DATA_BLOCK "DB11_INFORMES"
TITLE = DB11_INFORMES
{ S7_Optimized_Access := 'TRUE' }
AUTHOR : ABH
FAMILY : ZeusControl
VERSION : 1.0
NON_RETAIN
   VAR RETAIN
      Gestion { S7_SetPoint := 'False'} : "UDT_ZC_INF_GESTION";
      Registro { S7_SetPoint := 'False'} : "UDT_ZC_INF_DATOS";
      Buffer { S7_SetPoint := 'False'} : Array[0.."N_MAX_INF_BUFFER"] of "UDT_ZC_INF_DATOS";
   END_VAR


BEGIN
   Gestion.HabilitacionGeneral := TRUE;
   Gestion.EstadoConexion := TRUE;
   Gestion.OrdenIniciar := FALSE;
   Gestion.Etapa := 0;
   Gestion.SP_Tiempo := 10;
   Gestion.TiempoActual := 0;
   Gestion.NumeroMaxIntentos := 3;
   Gestion.Aviso.Registrar := FALSE;
   Gestion.Aviso.Estado := 0;
   Gestion.Aviso.NumeroIntentosActual := 0;
   Gestion.Datos.Registrar := 0;
   Gestion.Datos.Id := '';
   Gestion.Datos.Tipo := 0;
   Gestion.Datos.Codigo := '';
   Gestion.Datos.Fecha_1.Ano := 0;
   Gestion.Datos.Fecha_1.Mes := 0;
   Gestion.Datos.Fecha_1.Dia := 0;
   Gestion.Datos.Fecha_1.DiaSemana := 0;
   Gestion.Datos.Fecha_1.Hora := 0;
   Gestion.Datos.Fecha_1.Minuto := 0;
   Gestion.Datos.Fecha_1.Segundo := 0;
   Gestion.Datos.Fecha_1.NanoSegundo := 0;
   Gestion.Datos.Fecha_2.Ano := 0;
   Gestion.Datos.Fecha_2.Mes := 0;
   Gestion.Datos.Fecha_2.Dia := 0;
   Gestion.Datos.Fecha_2.DiaSemana := 0;
   Gestion.Datos.Fecha_2.Hora := 0;
   Gestion.Datos.Fecha_2.Minuto := 0;
   Gestion.Datos.Fecha_2.Segundo := 0;
   Gestion.Datos.Fecha_2.NanoSegundo := 0;
   Gestion.Datos.Fecha_3.Ano := 0;
   Gestion.Datos.Fecha_3.Mes := 0;
   Gestion.Datos.Fecha_3.Dia := 0;
   Gestion.Datos.Fecha_3.DiaSemana := 0;
   Gestion.Datos.Fecha_3.Hora := 0;
   Gestion.Datos.Fecha_3.Minuto := 0;
   Gestion.Datos.Fecha_3.Segundo := 0;
   Gestion.Datos.Fecha_3.NanoSegundo := 0;
   Gestion.Datos.String_1 := '';
   Gestion.Datos.String_2 := '';
   Gestion.Datos.String_3 := '';
   Gestion.Datos.String_4 := '';
   Gestion.Datos.String_5 := '';
   Gestion.Datos.String_6 := '';
   Gestion.Datos.String_7 := '';
   Gestion.Datos.String_8 := '';
   Gestion.Datos.String_9 := '';
   Gestion.Datos.String_10 := '';
   Gestion.Datos.Bool_1 := FALSE;
   Gestion.Datos.Bool_2 := FALSE;
   Gestion.Datos.Bool_3 := FALSE;
   Gestion.Datos.Bool_4 := FALSE;
   Gestion.Datos.Bool_5 := FALSE;
   Gestion.Datos.Bool_6 := FALSE;
   Gestion.Datos.Bool_7 := FALSE;
   Gestion.Datos.Bool_8 := FALSE;
   Gestion.Datos.Bool_9 := FALSE;
   Gestion.Datos.Bool_10 := FALSE;
   Gestion.Datos.Bool_11 := FALSE;
   Gestion.Datos.Bool_12 := FALSE;
   Gestion.Datos.Bool_13 := FALSE;
   Gestion.Datos.Bool_14 := FALSE;
   Gestion.Datos.Bool_15 := FALSE;
   Gestion.Datos.Bool_16 := FALSE;
   Gestion.Datos.Bool_17 := FALSE;
   Gestion.Datos.Bool_18 := FALSE;
   Gestion.Datos.Bool_19 := FALSE;
   Gestion.Datos.Bool_20 := FALSE;
   Gestion.Datos.Bool_21 := FALSE;
   Gestion.Datos.Bool_22 := FALSE;
   Gestion.Datos.Bool_23 := FALSE;
   Gestion.Datos.Bool_24 := FALSE;
   Gestion.Datos.Bool_25 := FALSE;
   Gestion.Datos.Bool_26 := FALSE;
   Gestion.Datos.Bool_27 := FALSE;
   Gestion.Datos.Bool_28 := FALSE;
   Gestion.Datos.Bool_29 := FALSE;
   Gestion.Datos.Bool_30 := FALSE;
   Gestion.Datos.Bool_31 := FALSE;
   Gestion.Datos.Bool_32 := FALSE;
   Gestion.Datos.Real_1 := 0.0;
   Gestion.Datos.Real_2 := 0.0;
   Gestion.Datos.Real_3 := 0.0;
   Gestion.Datos.Real_4 := 0.0;
   Gestion.Datos.Real_5 := 0.0;
   Gestion.Datos.Real_6 := 0.0;
   Gestion.Datos.Real_7 := 0.0;
   Gestion.Datos.Real_8 := 0.0;
   Gestion.Datos.Real_9 := 0.0;
   Gestion.Datos.Real_10 := 0.0;
   Gestion.Datos.Real_11 := 0.0;
   Gestion.Datos.Real_12 := 0.0;
   Gestion.Datos.Real_13 := 0.0;
   Gestion.Datos.Real_14 := 0.0;
   Gestion.Datos.Real_15 := 0.0;
   Gestion.Datos.Real_16 := 0.0;
   Gestion.Datos.Real_17 := 0.0;
   Gestion.Datos.Real_18 := 0.0;
   Gestion.Datos.Real_19 := 0.0;
   Gestion.Datos.Real_20 := 0.0;
   Gestion.Datos.Int_1 := 0;
   Gestion.Datos.Int_2 := 0;
   Gestion.Datos.Int_3 := 0;
   Gestion.Datos.Int_4 := 0;
   Gestion.Datos.Int_5 := 0;
   Gestion.Datos.Int_6 := 0;
   Gestion.Datos.Int_7 := 0;
   Gestion.Datos.Int_8 := 0;
   Gestion.Datos.Int_9 := 0;
   Gestion.Datos.Int_10 := 0;
   Gestion.Datos.Int_11 := 0;
   Gestion.Datos.Int_12 := 0;
   Gestion.Datos.Int_13 := 0;
   Gestion.Datos.Int_14 := 0;
   Gestion.Datos.Int_15 := 0;
   Gestion.Datos.Int_16 := 0;
   Gestion.Datos.Int_17 := 0;
   Gestion.Datos.Int_18 := 0;
   Gestion.Datos.Int_19 := 0;
   Gestion.Datos.Int_20 := 0;
   Registro.Registrar := 0;
   Registro.Id := '';
   Registro.Tipo := 0;
   Registro.Codigo := '';
   Registro.Fecha_1.Ano := 0;
   Registro.Fecha_1.Mes := 0;
   Registro.Fecha_1.Dia := 0;
   Registro.Fecha_1.DiaSemana := 0;
   Registro.Fecha_1.Hora := 0;
   Registro.Fecha_1.Minuto := 0;
   Registro.Fecha_1.Segundo := 0;
   Registro.Fecha_1.NanoSegundo := 0;
   Registro.Fecha_2.Ano := 0;
   Registro.Fecha_2.Mes := 0;
   Registro.Fecha_2.Dia := 0;
   Registro.Fecha_2.DiaSemana := 0;
   Registro.Fecha_2.Hora := 0;
   Registro.Fecha_2.Minuto := 0;
   Registro.Fecha_2.Segundo := 0;
   Registro.Fecha_2.NanoSegundo := 0;
   Registro.Fecha_3.Ano := 0;
   Registro.Fecha_3.Mes := 0;
   Registro.Fecha_3.Dia := 0;
   Registro.Fecha_3.DiaSemana := 0;
   Registro.Fecha_3.Hora := 0;
   Registro.Fecha_3.Minuto := 0;
   Registro.Fecha_3.Segundo := 0;
   Registro.Fecha_3.NanoSegundo := 0;
   Registro.String_1 := '';
   Registro.String_2 := '';
   Registro.String_3 := '';
   Registro.String_4 := '';
   Registro.String_5 := '';
   Registro.String_6 := '';
   Registro.String_7 := '';
   Registro.String_8 := '';
   Registro.String_9 := '';
   Registro.String_10 := '';
   Registro.Bool_1 := FALSE;
   Registro.Bool_2 := FALSE;
   Registro.Bool_3 := FALSE;
   Registro.Bool_4 := FALSE;
   Registro.Bool_5 := FALSE;
   Registro.Bool_6 := FALSE;
   Registro.Bool_7 := FALSE;
   Registro.Bool_8 := FALSE;
   Registro.Bool_9 := FALSE;
   Registro.Bool_10 := FALSE;
   Registro.Bool_11 := FALSE;
   Registro.Bool_12 := FALSE;
   Registro.Bool_13 := FALSE;
   Registro.Bool_14 := FALSE;
   Registro.Bool_15 := FALSE;
   Registro.Bool_16 := FALSE;
   Registro.Bool_17 := FALSE;
   Registro.Bool_18 := FALSE;
   Registro.Bool_19 := FALSE;
   Registro.Bool_20 := FALSE;
   Registro.Bool_21 := FALSE;
   Registro.Bool_22 := FALSE;
   Registro.Bool_23 := FALSE;
   Registro.Bool_24 := FALSE;
   Registro.Bool_25 := FALSE;
   Registro.Bool_26 := FALSE;
   Registro.Bool_27 := FALSE;
   Registro.Bool_28 := FALSE;
   Registro.Bool_29 := FALSE;
   Registro.Bool_30 := FALSE;
   Registro.Bool_31 := FALSE;
   Registro.Bool_32 := FALSE;
   Registro.Real_1 := 0.0;
   Registro.Real_2 := 0.0;
   Registro.Real_3 := 0.0;
   Registro.Real_4 := 0.0;
   Registro.Real_5 := 0.0;
   Registro.Real_6 := 0.0;
   Registro.Real_7 := 0.0;
   Registro.Real_8 := 0.0;
   Registro.Real_9 := 0.0;
   Registro.Real_10 := 0.0;
   Registro.Real_11 := 0.0;
   Registro.Real_12 := 0.0;
   Registro.Real_13 := 0.0;
   Registro.Real_14 := 0.0;
   Registro.Real_15 := 0.0;
   Registro.Real_16 := 0.0;
   Registro.Real_17 := 0.0;
   Registro.Real_18 := 0.0;
   Registro.Real_19 := 0.0;
   Registro.Real_20 := 0.0;
   Registro.Int_1 := 0;
   Registro.Int_2 := 0;
   Registro.Int_3 := 0;
   Registro.Int_4 := 0;
   Registro.Int_5 := 0;
   Registro.Int_6 := 0;
   Registro.Int_7 := 0;
   Registro.Int_8 := 0;
   Registro.Int_9 := 0;
   Registro.Int_10 := 0;
   Registro.Int_11 := 0;
   Registro.Int_12 := 0;
   Registro.Int_13 := 0;
   Registro.Int_14 := 0;
   Registro.Int_15 := 0;
   Registro.Int_16 := 0;
   Registro.Int_17 := 0;
   Registro.Int_18 := 0;
   Registro.Int_19 := 0;
   Registro.Int_20 := 0;
   Buffer[0].Registrar := 0;
   Buffer[0].Id := '';
   Buffer[0].Tipo := 0;
   Buffer[0].Codigo := '';
   Buffer[0].Fecha_1.Ano := 0;
   Buffer[0].Fecha_1.Mes := 0;
   Buffer[0].Fecha_1.Dia := 0;
   Buffer[0].Fecha_1.DiaSemana := 0;
   Buffer[0].Fecha_1.Hora := 0;
   Buffer[0].Fecha_1.Minuto := 0;
   Buffer[0].Fecha_1.Segundo := 0;
   Buffer[0].Fecha_1.NanoSegundo := 0;
   Buffer[0].Fecha_2.Ano := 0;
   Buffer[0].Fecha_2.Mes := 0;
   Buffer[0].Fecha_2.Dia := 0;
   Buffer[0].Fecha_2.DiaSemana := 0;
   Buffer[0].Fecha_2.Hora := 0;
   Buffer[0].Fecha_2.Minuto := 0;
   Buffer[0].Fecha_2.Segundo := 0;
   Buffer[0].Fecha_2.NanoSegundo := 0;
   Buffer[0].Fecha_3.Ano := 0;
   Buffer[0].Fecha_3.Mes := 0;
   Buffer[0].Fecha_3.Dia := 0;
   Buffer[0].Fecha_3.DiaSemana := 0;
   Buffer[0].Fecha_3.Hora := 0;
   Buffer[0].Fecha_3.Minuto := 0;
   Buffer[0].Fecha_3.Segundo := 0;
   Buffer[0].Fecha_3.NanoSegundo := 0;
   Buffer[0].String_1 := '';
   Buffer[0].String_2 := '';
   Buffer[0].String_3 := '';
   Buffer[0].String_4 := '';
   Buffer[0].String_5 := '';
   Buffer[0].String_6 := '';
   Buffer[0].String_7 := '';
   Buffer[0].String_8 := '';
   Buffer[0].String_9 := '';
   Buffer[0].String_10 := '';
   Buffer[0].Bool_1 := FALSE;
   Buffer[0].Bool_2 := FALSE;
   Buffer[0].Bool_3 := FALSE;
   Buffer[0].Bool_4 := FALSE;
   Buffer[0].Bool_5 := FALSE;
   Buffer[0].Bool_6 := FALSE;
   Buffer[0].Bool_7 := FALSE;
   Buffer[0].Bool_8 := FALSE;
   Buffer[0].Bool_9 := FALSE;
   Buffer[0].Bool_10 := FALSE;
   Buffer[0].Bool_11 := FALSE;
   Buffer[0].Bool_12 := FALSE;
   Buffer[0].Bool_13 := FALSE;
   Buffer[0].Bool_14 := FALSE;
   Buffer[0].Bool_15 := FALSE;
   Buffer[0].Bool_16 := FALSE;
   Buffer[0].Bool_17 := FALSE;
   Buffer[0].Bool_18 := FALSE;
   Buffer[0].Bool_19 := FALSE;
   Buffer[0].Bool_20 := FALSE;
   Buffer[0].Bool_21 := FALSE;
   Buffer[0].Bool_22 := FALSE;
   Buffer[0].Bool_23 := FALSE;
   Buffer[0].Bool_24 := FALSE;
   Buffer[0].Bool_25 := FALSE;
   Buffer[0].Bool_26 := FALSE;
   Buffer[0].Bool_27 := FALSE;
   Buffer[0].Bool_28 := FALSE;
   Buffer[0].Bool_29 := FALSE;
   Buffer[0].Bool_30 := FALSE;
   Buffer[0].Bool_31 := FALSE;
   Buffer[0].Bool_32 := FALSE;
   Buffer[0].Real_1 := 0.0;
   Buffer[0].Real_2 := 0.0;
   Buffer[0].Real_3 := 0.0;
   Buffer[0].Real_4 := 0.0;
   Buffer[0].Real_5 := 0.0;
   Buffer[0].Real_6 := 0.0;
   Buffer[0].Real_7 := 0.0;
   Buffer[0].Real_8 := 0.0;
   Buffer[0].Real_9 := 0.0;
   Buffer[0].Real_10 := 0.0;
   Buffer[0].Real_11 := 0.0;
   Buffer[0].Real_12 := 0.0;
   Buffer[0].Real_13 := 0.0;
   Buffer[0].Real_14 := 0.0;
   Buffer[0].Real_15 := 0.0;
   Buffer[0].Real_16 := 0.0;
   Buffer[0].Real_17 := 0.0;
   Buffer[0].Real_18 := 0.0;
   Buffer[0].Real_19 := 0.0;
   Buffer[0].Real_20 := 0.0;
   Buffer[0].Int_1 := 0;
   Buffer[0].Int_2 := 0;
   Buffer[0].Int_3 := 0;
   Buffer[0].Int_4 := 0;
   Buffer[0].Int_5 := 0;
   Buffer[0].Int_6 := 0;
   Buffer[0].Int_7 := 0;
   Buffer[0].Int_8 := 0;
   Buffer[0].Int_9 := 0;
   Buffer[0].Int_10 := 0;
   Buffer[0].Int_11 := 0;
   Buffer[0].Int_12 := 0;
   Buffer[0].Int_13 := 0;
   Buffer[0].Int_14 := 0;
   Buffer[0].Int_15 := 0;
   Buffer[0].Int_16 := 0;
   Buffer[0].Int_17 := 0;
   Buffer[0].Int_18 := 0;
   Buffer[0].Int_19 := 0;
   Buffer[0].Int_20 := 0;
   Buffer[1].Registrar := 0;
   Buffer[1].Id := '';
   Buffer[1].Tipo := 0;
   Buffer[1].Codigo := '';
   Buffer[1].Fecha_1.Ano := 0;
   Buffer[1].Fecha_1.Mes := 0;
   Buffer[1].Fecha_1.Dia := 0;
   Buffer[1].Fecha_1.DiaSemana := 0;
   Buffer[1].Fecha_1.Hora := 0;
   Buffer[1].Fecha_1.Minuto := 0;
   Buffer[1].Fecha_1.Segundo := 0;
   Buffer[1].Fecha_1.NanoSegundo := 0;
   Buffer[1].Fecha_2.Ano := 0;
   Buffer[1].Fecha_2.Mes := 0;
   Buffer[1].Fecha_2.Dia := 0;
   Buffer[1].Fecha_2.DiaSemana := 0;
   Buffer[1].Fecha_2.Hora := 0;
   Buffer[1].Fecha_2.Minuto := 0;
   Buffer[1].Fecha_2.Segundo := 0;
   Buffer[1].Fecha_2.NanoSegundo := 0;
   Buffer[1].Fecha_3.Ano := 0;
   Buffer[1].Fecha_3.Mes := 0;
   Buffer[1].Fecha_3.Dia := 0;
   Buffer[1].Fecha_3.DiaSemana := 0;
   Buffer[1].Fecha_3.Hora := 0;
   Buffer[1].Fecha_3.Minuto := 0;
   Buffer[1].Fecha_3.Segundo := 0;
   Buffer[1].Fecha_3.NanoSegundo := 0;
   Buffer[1].String_1 := '';
   Buffer[1].String_2 := '';
   Buffer[1].String_3 := '';
   Buffer[1].String_4 := '';
   Buffer[1].String_5 := '';
   Buffer[1].String_6 := '';
   Buffer[1].String_7 := '';
   Buffer[1].String_8 := '';
   Buffer[1].String_9 := '';
   Buffer[1].String_10 := '';
   Buffer[1].Bool_1 := FALSE;
   Buffer[1].Bool_2 := FALSE;
   Buffer[1].Bool_3 := FALSE;
   Buffer[1].Bool_4 := FALSE;
   Buffer[1].Bool_5 := FALSE;
   Buffer[1].Bool_6 := FALSE;
   Buffer[1].Bool_7 := FALSE;
   Buffer[1].Bool_8 := FALSE;
   Buffer[1].Bool_9 := FALSE;
   Buffer[1].Bool_10 := FALSE;
   Buffer[1].Bool_11 := FALSE;
   Buffer[1].Bool_12 := FALSE;
   Buffer[1].Bool_13 := FALSE;
   Buffer[1].Bool_14 := FALSE;
   Buffer[1].Bool_15 := FALSE;
   Buffer[1].Bool_16 := FALSE;
   Buffer[1].Bool_17 := FALSE;
   Buffer[1].Bool_18 := FALSE;
   Buffer[1].Bool_19 := FALSE;
   Buffer[1].Bool_20 := FALSE;
   Buffer[1].Bool_21 := FALSE;
   Buffer[1].Bool_22 := FALSE;
   Buffer[1].Bool_23 := FALSE;
   Buffer[1].Bool_24 := FALSE;
   Buffer[1].Bool_25 := FALSE;
   Buffer[1].Bool_26 := FALSE;
   Buffer[1].Bool_27 := FALSE;
   Buffer[1].Bool_28 := FALSE;
   Buffer[1].Bool_29 := FALSE;
   Buffer[1].Bool_30 := FALSE;
   Buffer[1].Bool_31 := FALSE;
   Buffer[1].Bool_32 := FALSE;
   Buffer[1].Real_1 := 0.0;
   Buffer[1].Real_2 := 0.0;
   Buffer[1].Real_3 := 0.0;
   Buffer[1].Real_4 := 0.0;
   Buffer[1].Real_5 := 0.0;
   Buffer[1].Real_6 := 0.0;
   Buffer[1].Real_7 := 0.0;
   Buffer[1].Real_8 := 0.0;
   Buffer[1].Real_9 := 0.0;
   Buffer[1].Real_10 := 0.0;
   Buffer[1].Real_11 := 0.0;
   Buffer[1].Real_12 := 0.0;
   Buffer[1].Real_13 := 0.0;
   Buffer[1].Real_14 := 0.0;
   Buffer[1].Real_15 := 0.0;
   Buffer[1].Real_16 := 0.0;
   Buffer[1].Real_17 := 0.0;
   Buffer[1].Real_18 := 0.0;
   Buffer[1].Real_19 := 0.0;
   Buffer[1].Real_20 := 0.0;
   Buffer[1].Int_1 := 0;
   Buffer[1].Int_2 := 0;
   Buffer[1].Int_3 := 0;
   Buffer[1].Int_4 := 0;
   Buffer[1].Int_5 := 0;
   Buffer[1].Int_6 := 0;
   Buffer[1].Int_7 := 0;
   Buffer[1].Int_8 := 0;
   Buffer[1].Int_9 := 0;
   Buffer[1].Int_10 := 0;
   Buffer[1].Int_11 := 0;
   Buffer[1].Int_12 := 0;
   Buffer[1].Int_13 := 0;
   Buffer[1].Int_14 := 0;
   Buffer[1].Int_15 := 0;
   Buffer[1].Int_16 := 0;
   Buffer[1].Int_17 := 0;
   Buffer[1].Int_18 := 0;
   Buffer[1].Int_19 := 0;
   Buffer[1].Int_20 := 0;
   Buffer[2].Registrar := 0;
   Buffer[2].Id := '';
   Buffer[2].Tipo := 0;
   Buffer[2].Codigo := '';
   Buffer[2].Fecha_1.Ano := 0;
   Buffer[2].Fecha_1.Mes := 0;
   Buffer[2].Fecha_1.Dia := 0;
   Buffer[2].Fecha_1.DiaSemana := 0;
   Buffer[2].Fecha_1.Hora := 0;
   Buffer[2].Fecha_1.Minuto := 0;
   Buffer[2].Fecha_1.Segundo := 0;
   Buffer[2].Fecha_1.NanoSegundo := 0;
   Buffer[2].Fecha_2.Ano := 0;
   Buffer[2].Fecha_2.Mes := 0;
   Buffer[2].Fecha_2.Dia := 0;
   Buffer[2].Fecha_2.DiaSemana := 0;
   Buffer[2].Fecha_2.Hora := 0;
   Buffer[2].Fecha_2.Minuto := 0;
   Buffer[2].Fecha_2.Segundo := 0;
   Buffer[2].Fecha_2.NanoSegundo := 0;
   Buffer[2].Fecha_3.Ano := 0;
   Buffer[2].Fecha_3.Mes := 0;
   Buffer[2].Fecha_3.Dia := 0;
   Buffer[2].Fecha_3.DiaSemana := 0;
   Buffer[2].Fecha_3.Hora := 0;
   Buffer[2].Fecha_3.Minuto := 0;
   Buffer[2].Fecha_3.Segundo := 0;
   Buffer[2].Fecha_3.NanoSegundo := 0;
   Buffer[2].String_1 := '';
   Buffer[2].String_2 := '';
   Buffer[2].String_3 := '';
   Buffer[2].String_4 := '';
   Buffer[2].String_5 := '';
   Buffer[2].String_6 := '';
   Buffer[2].String_7 := '';
   Buffer[2].String_8 := '';
   Buffer[2].String_9 := '';
   Buffer[2].String_10 := '';
   Buffer[2].Bool_1 := FALSE;
   Buffer[2].Bool_2 := FALSE;
   Buffer[2].Bool_3 := FALSE;
   Buffer[2].Bool_4 := FALSE;
   Buffer[2].Bool_5 := FALSE;
   Buffer[2].Bool_6 := FALSE;
   Buffer[2].Bool_7 := FALSE;
   Buffer[2].Bool_8 := FALSE;
   Buffer[2].Bool_9 := FALSE;
   Buffer[2].Bool_10 := FALSE;
   Buffer[2].Bool_11 := FALSE;
   Buffer[2].Bool_12 := FALSE;
   Buffer[2].Bool_13 := FALSE;
   Buffer[2].Bool_14 := FALSE;
   Buffer[2].Bool_15 := FALSE;
   Buffer[2].Bool_16 := FALSE;
   Buffer[2].Bool_17 := FALSE;
   Buffer[2].Bool_18 := FALSE;
   Buffer[2].Bool_19 := FALSE;
   Buffer[2].Bool_20 := FALSE;
   Buffer[2].Bool_21 := FALSE;
   Buffer[2].Bool_22 := FALSE;
   Buffer[2].Bool_23 := FALSE;
   Buffer[2].Bool_24 := FALSE;
   Buffer[2].Bool_25 := FALSE;
   Buffer[2].Bool_26 := FALSE;
   Buffer[2].Bool_27 := FALSE;
   Buffer[2].Bool_28 := FALSE;
   Buffer[2].Bool_29 := FALSE;
   Buffer[2].Bool_30 := FALSE;
   Buffer[2].Bool_31 := FALSE;
   Buffer[2].Bool_32 := FALSE;
   Buffer[2].Real_1 := 0.0;
   Buffer[2].Real_2 := 0.0;
   Buffer[2].Real_3 := 0.0;
   Buffer[2].Real_4 := 0.0;
   Buffer[2].Real_5 := 0.0;
   Buffer[2].Real_6 := 0.0;
   Buffer[2].Real_7 := 0.0;
   Buffer[2].Real_8 := 0.0;
   Buffer[2].Real_9 := 0.0;
   Buffer[2].Real_10 := 0.0;
   Buffer[2].Real_11 := 0.0;
   Buffer[2].Real_12 := 0.0;
   Buffer[2].Real_13 := 0.0;
   Buffer[2].Real_14 := 0.0;
   Buffer[2].Real_15 := 0.0;
   Buffer[2].Real_16 := 0.0;
   Buffer[2].Real_17 := 0.0;
   Buffer[2].Real_18 := 0.0;
   Buffer[2].Real_19 := 0.0;
   Buffer[2].Real_20 := 0.0;
   Buffer[2].Int_1 := 0;
   Buffer[2].Int_2 := 0;
   Buffer[2].Int_3 := 0;
   Buffer[2].Int_4 := 0;
   Buffer[2].Int_5 := 0;
   Buffer[2].Int_6 := 0;
   Buffer[2].Int_7 := 0;
   Buffer[2].Int_8 := 0;
   Buffer[2].Int_9 := 0;
   Buffer[2].Int_10 := 0;
   Buffer[2].Int_11 := 0;
   Buffer[2].Int_12 := 0;
   Buffer[2].Int_13 := 0;
   Buffer[2].Int_14 := 0;
   Buffer[2].Int_15 := 0;
   Buffer[2].Int_16 := 0;
   Buffer[2].Int_17 := 0;
   Buffer[2].Int_18 := 0;
   Buffer[2].Int_19 := 0;
   Buffer[2].Int_20 := 0;
   Buffer[3].Registrar := 0;
   Buffer[3].Id := '';
   Buffer[3].Tipo := 0;
   Buffer[3].Codigo := '';
   Buffer[3].Fecha_1.Ano := 0;
   Buffer[3].Fecha_1.Mes := 0;
   Buffer[3].Fecha_1.Dia := 0;
   Buffer[3].Fecha_1.DiaSemana := 0;
   Buffer[3].Fecha_1.Hora := 0;
   Buffer[3].Fecha_1.Minuto := 0;
   Buffer[3].Fecha_1.Segundo := 0;
   Buffer[3].Fecha_1.NanoSegundo := 0;
   Buffer[3].Fecha_2.Ano := 0;
   Buffer[3].Fecha_2.Mes := 0;
   Buffer[3].Fecha_2.Dia := 0;
   Buffer[3].Fecha_2.DiaSemana := 0;
   Buffer[3].Fecha_2.Hora := 0;
   Buffer[3].Fecha_2.Minuto := 0;
   Buffer[3].Fecha_2.Segundo := 0;
   Buffer[3].Fecha_2.NanoSegundo := 0;
   Buffer[3].Fecha_3.Ano := 0;
   Buffer[3].Fecha_3.Mes := 0;
   Buffer[3].Fecha_3.Dia := 0;
   Buffer[3].Fecha_3.DiaSemana := 0;
   Buffer[3].Fecha_3.Hora := 0;
   Buffer[3].Fecha_3.Minuto := 0;
   Buffer[3].Fecha_3.Segundo := 0;
   Buffer[3].Fecha_3.NanoSegundo := 0;
   Buffer[3].String_1 := '';
   Buffer[3].String_2 := '';
   Buffer[3].String_3 := '';
   Buffer[3].String_4 := '';
   Buffer[3].String_5 := '';
   Buffer[3].String_6 := '';
   Buffer[3].String_7 := '';
   Buffer[3].String_8 := '';
   Buffer[3].String_9 := '';
   Buffer[3].String_10 := '';
   Buffer[3].Bool_1 := FALSE;
   Buffer[3].Bool_2 := FALSE;
   Buffer[3].Bool_3 := FALSE;
   Buffer[3].Bool_4 := FALSE;
   Buffer[3].Bool_5 := FALSE;
   Buffer[3].Bool_6 := FALSE;
   Buffer[3].Bool_7 := FALSE;
   Buffer[3].Bool_8 := FALSE;
   Buffer[3].Bool_9 := FALSE;
   Buffer[3].Bool_10 := FALSE;
   Buffer[3].Bool_11 := FALSE;
   Buffer[3].Bool_12 := FALSE;
   Buffer[3].Bool_13 := FALSE;
   Buffer[3].Bool_14 := FALSE;
   Buffer[3].Bool_15 := FALSE;
   Buffer[3].Bool_16 := FALSE;
   Buffer[3].Bool_17 := FALSE;
   Buffer[3].Bool_18 := FALSE;
   Buffer[3].Bool_19 := FALSE;
   Buffer[3].Bool_20 := FALSE;
   Buffer[3].Bool_21 := FALSE;
   Buffer[3].Bool_22 := FALSE;
   Buffer[3].Bool_23 := FALSE;
   Buffer[3].Bool_24 := FALSE;
   Buffer[3].Bool_25 := FALSE;
   Buffer[3].Bool_26 := FALSE;
   Buffer[3].Bool_27 := FALSE;
   Buffer[3].Bool_28 := FALSE;
   Buffer[3].Bool_29 := FALSE;
   Buffer[3].Bool_30 := FALSE;
   Buffer[3].Bool_31 := FALSE;
   Buffer[3].Bool_32 := FALSE;
   Buffer[3].Real_1 := 0.0;
   Buffer[3].Real_2 := 0.0;
   Buffer[3].Real_3 := 0.0;
   Buffer[3].Real_4 := 0.0;
   Buffer[3].Real_5 := 0.0;
   Buffer[3].Real_6 := 0.0;
   Buffer[3].Real_7 := 0.0;
   Buffer[3].Real_8 := 0.0;
   Buffer[3].Real_9 := 0.0;
   Buffer[3].Real_10 := 0.0;
   Buffer[3].Real_11 := 0.0;
   Buffer[3].Real_12 := 0.0;
   Buffer[3].Real_13 := 0.0;
   Buffer[3].Real_14 := 0.0;
   Buffer[3].Real_15 := 0.0;
   Buffer[3].Real_16 := 0.0;
   Buffer[3].Real_17 := 0.0;
   Buffer[3].Real_18 := 0.0;
   Buffer[3].Real_19 := 0.0;
   Buffer[3].Real_20 := 0.0;
   Buffer[3].Int_1 := 0;
   Buffer[3].Int_2 := 0;
   Buffer[3].Int_3 := 0;
   Buffer[3].Int_4 := 0;
   Buffer[3].Int_5 := 0;
   Buffer[3].Int_6 := 0;
   Buffer[3].Int_7 := 0;
   Buffer[3].Int_8 := 0;
   Buffer[3].Int_9 := 0;
   Buffer[3].Int_10 := 0;
   Buffer[3].Int_11 := 0;
   Buffer[3].Int_12 := 0;
   Buffer[3].Int_13 := 0;
   Buffer[3].Int_14 := 0;
   Buffer[3].Int_15 := 0;
   Buffer[3].Int_16 := 0;
   Buffer[3].Int_17 := 0;
   Buffer[3].Int_18 := 0;
   Buffer[3].Int_19 := 0;
   Buffer[3].Int_20 := 0;
   Buffer[4].Registrar := 0;
   Buffer[4].Id := '';
   Buffer[4].Tipo := 0;
   Buffer[4].Codigo := '';
   Buffer[4].Fecha_1.Ano := 0;
   Buffer[4].Fecha_1.Mes := 0;
   Buffer[4].Fecha_1.Dia := 0;
   Buffer[4].Fecha_1.DiaSemana := 0;
   Buffer[4].Fecha_1.Hora := 0;
   Buffer[4].Fecha_1.Minuto := 0;
   Buffer[4].Fecha_1.Segundo := 0;
   Buffer[4].Fecha_1.NanoSegundo := 0;
   Buffer[4].Fecha_2.Ano := 0;
   Buffer[4].Fecha_2.Mes := 0;
   Buffer[4].Fecha_2.Dia := 0;
   Buffer[4].Fecha_2.DiaSemana := 0;
   Buffer[4].Fecha_2.Hora := 0;
   Buffer[4].Fecha_2.Minuto := 0;
   Buffer[4].Fecha_2.Segundo := 0;
   Buffer[4].Fecha_2.NanoSegundo := 0;
   Buffer[4].Fecha_3.Ano := 0;
   Buffer[4].Fecha_3.Mes := 0;
   Buffer[4].Fecha_3.Dia := 0;
   Buffer[4].Fecha_3.DiaSemana := 0;
   Buffer[4].Fecha_3.Hora := 0;
   Buffer[4].Fecha_3.Minuto := 0;
   Buffer[4].Fecha_3.Segundo := 0;
   Buffer[4].Fecha_3.NanoSegundo := 0;
   Buffer[4].String_1 := '';
   Buffer[4].String_2 := '';
   Buffer[4].String_3 := '';
   Buffer[4].String_4 := '';
   Buffer[4].String_5 := '';
   Buffer[4].String_6 := '';
   Buffer[4].String_7 := '';
   Buffer[4].String_8 := '';
   Buffer[4].String_9 := '';
   Buffer[4].String_10 := '';
   Buffer[4].Bool_1 := FALSE;
   Buffer[4].Bool_2 := FALSE;
   Buffer[4].Bool_3 := FALSE;
   Buffer[4].Bool_4 := FALSE;
   Buffer[4].Bool_5 := FALSE;
   Buffer[4].Bool_6 := FALSE;
   Buffer[4].Bool_7 := FALSE;
   Buffer[4].Bool_8 := FALSE;
   Buffer[4].Bool_9 := FALSE;
   Buffer[4].Bool_10 := FALSE;
   Buffer[4].Bool_11 := FALSE;
   Buffer[4].Bool_12 := FALSE;
   Buffer[4].Bool_13 := FALSE;
   Buffer[4].Bool_14 := FALSE;
   Buffer[4].Bool_15 := FALSE;
   Buffer[4].Bool_16 := FALSE;
   Buffer[4].Bool_17 := FALSE;
   Buffer[4].Bool_18 := FALSE;
   Buffer[4].Bool_19 := FALSE;
   Buffer[4].Bool_20 := FALSE;
   Buffer[4].Bool_21 := FALSE;
   Buffer[4].Bool_22 := FALSE;
   Buffer[4].Bool_23 := FALSE;
   Buffer[4].Bool_24 := FALSE;
   Buffer[4].Bool_25 := FALSE;
   Buffer[4].Bool_26 := FALSE;
   Buffer[4].Bool_27 := FALSE;
   Buffer[4].Bool_28 := FALSE;
   Buffer[4].Bool_29 := FALSE;
   Buffer[4].Bool_30 := FALSE;
   Buffer[4].Bool_31 := FALSE;
   Buffer[4].Bool_32 := FALSE;
   Buffer[4].Real_1 := 0.0;
   Buffer[4].Real_2 := 0.0;
   Buffer[4].Real_3 := 0.0;
   Buffer[4].Real_4 := 0.0;
   Buffer[4].Real_5 := 0.0;
   Buffer[4].Real_6 := 0.0;
   Buffer[4].Real_7 := 0.0;
   Buffer[4].Real_8 := 0.0;
   Buffer[4].Real_9 := 0.0;
   Buffer[4].Real_10 := 0.0;
   Buffer[4].Real_11 := 0.0;
   Buffer[4].Real_12 := 0.0;
   Buffer[4].Real_13 := 0.0;
   Buffer[4].Real_14 := 0.0;
   Buffer[4].Real_15 := 0.0;
   Buffer[4].Real_16 := 0.0;
   Buffer[4].Real_17 := 0.0;
   Buffer[4].Real_18 := 0.0;
   Buffer[4].Real_19 := 0.0;
   Buffer[4].Real_20 := 0.0;
   Buffer[4].Int_1 := 0;
   Buffer[4].Int_2 := 0;
   Buffer[4].Int_3 := 0;
   Buffer[4].Int_4 := 0;
   Buffer[4].Int_5 := 0;
   Buffer[4].Int_6 := 0;
   Buffer[4].Int_7 := 0;
   Buffer[4].Int_8 := 0;
   Buffer[4].Int_9 := 0;
   Buffer[4].Int_10 := 0;
   Buffer[4].Int_11 := 0;
   Buffer[4].Int_12 := 0;
   Buffer[4].Int_13 := 0;
   Buffer[4].Int_14 := 0;
   Buffer[4].Int_15 := 0;
   Buffer[4].Int_16 := 0;
   Buffer[4].Int_17 := 0;
   Buffer[4].Int_18 := 0;
   Buffer[4].Int_19 := 0;
   Buffer[4].Int_20 := 0;
   Buffer[5].Registrar := 0;
   Buffer[5].Id := '';
   Buffer[5].Tipo := 0;
   Buffer[5].Codigo := '';
   Buffer[5].Fecha_1.Ano := 0;
   Buffer[5].Fecha_1.Mes := 0;
   Buffer[5].Fecha_1.Dia := 0;
   Buffer[5].Fecha_1.DiaSemana := 0;
   Buffer[5].Fecha_1.Hora := 0;
   Buffer[5].Fecha_1.Minuto := 0;
   Buffer[5].Fecha_1.Segundo := 0;
   Buffer[5].Fecha_1.NanoSegundo := 0;
   Buffer[5].Fecha_2.Ano := 0;
   Buffer[5].Fecha_2.Mes := 0;
   Buffer[5].Fecha_2.Dia := 0;
   Buffer[5].Fecha_2.DiaSemana := 0;
   Buffer[5].Fecha_2.Hora := 0;
   Buffer[5].Fecha_2.Minuto := 0;
   Buffer[5].Fecha_2.Segundo := 0;
   Buffer[5].Fecha_2.NanoSegundo := 0;
   Buffer[5].Fecha_3.Ano := 0;
   Buffer[5].Fecha_3.Mes := 0;
   Buffer[5].Fecha_3.Dia := 0;
   Buffer[5].Fecha_3.DiaSemana := 0;
   Buffer[5].Fecha_3.Hora := 0;
   Buffer[5].Fecha_3.Minuto := 0;
   Buffer[5].Fecha_3.Segundo := 0;
   Buffer[5].Fecha_3.NanoSegundo := 0;
   Buffer[5].String_1 := '';
   Buffer[5].String_2 := '';
   Buffer[5].String_3 := '';
   Buffer[5].String_4 := '';
   Buffer[5].String_5 := '';
   Buffer[5].String_6 := '';
   Buffer[5].String_7 := '';
   Buffer[5].String_8 := '';
   Buffer[5].String_9 := '';
   Buffer[5].String_10 := '';
   Buffer[5].Bool_1 := FALSE;
   Buffer[5].Bool_2 := FALSE;
   Buffer[5].Bool_3 := FALSE;
   Buffer[5].Bool_4 := FALSE;
   Buffer[5].Bool_5 := FALSE;
   Buffer[5].Bool_6 := FALSE;
   Buffer[5].Bool_7 := FALSE;
   Buffer[5].Bool_8 := FALSE;
   Buffer[5].Bool_9 := FALSE;
   Buffer[5].Bool_10 := FALSE;
   Buffer[5].Bool_11 := FALSE;
   Buffer[5].Bool_12 := FALSE;
   Buffer[5].Bool_13 := FALSE;
   Buffer[5].Bool_14 := FALSE;
   Buffer[5].Bool_15 := FALSE;
   Buffer[5].Bool_16 := FALSE;
   Buffer[5].Bool_17 := FALSE;
   Buffer[5].Bool_18 := FALSE;
   Buffer[5].Bool_19 := FALSE;
   Buffer[5].Bool_20 := FALSE;
   Buffer[5].Bool_21 := FALSE;
   Buffer[5].Bool_22 := FALSE;
   Buffer[5].Bool_23 := FALSE;
   Buffer[5].Bool_24 := FALSE;
   Buffer[5].Bool_25 := FALSE;
   Buffer[5].Bool_26 := FALSE;
   Buffer[5].Bool_27 := FALSE;
   Buffer[5].Bool_28 := FALSE;
   Buffer[5].Bool_29 := FALSE;
   Buffer[5].Bool_30 := FALSE;
   Buffer[5].Bool_31 := FALSE;
   Buffer[5].Bool_32 := FALSE;
   Buffer[5].Real_1 := 0.0;
   Buffer[5].Real_2 := 0.0;
   Buffer[5].Real_3 := 0.0;
   Buffer[5].Real_4 := 0.0;
   Buffer[5].Real_5 := 0.0;
   Buffer[5].Real_6 := 0.0;
   Buffer[5].Real_7 := 0.0;
   Buffer[5].Real_8 := 0.0;
   Buffer[5].Real_9 := 0.0;
   Buffer[5].Real_10 := 0.0;
   Buffer[5].Real_11 := 0.0;
   Buffer[5].Real_12 := 0.0;
   Buffer[5].Real_13 := 0.0;
   Buffer[5].Real_14 := 0.0;
   Buffer[5].Real_15 := 0.0;
   Buffer[5].Real_16 := 0.0;
   Buffer[5].Real_17 := 0.0;
   Buffer[5].Real_18 := 0.0;
   Buffer[5].Real_19 := 0.0;
   Buffer[5].Real_20 := 0.0;
   Buffer[5].Int_1 := 0;
   Buffer[5].Int_2 := 0;
   Buffer[5].Int_3 := 0;
   Buffer[5].Int_4 := 0;
   Buffer[5].Int_5 := 0;
   Buffer[5].Int_6 := 0;
   Buffer[5].Int_7 := 0;
   Buffer[5].Int_8 := 0;
   Buffer[5].Int_9 := 0;
   Buffer[5].Int_10 := 0;
   Buffer[5].Int_11 := 0;
   Buffer[5].Int_12 := 0;
   Buffer[5].Int_13 := 0;
   Buffer[5].Int_14 := 0;
   Buffer[5].Int_15 := 0;
   Buffer[5].Int_16 := 0;
   Buffer[5].Int_17 := 0;
   Buffer[5].Int_18 := 0;
   Buffer[5].Int_19 := 0;
   Buffer[5].Int_20 := 0;
   Buffer[6].Registrar := 0;
   Buffer[6].Id := '';
   Buffer[6].Tipo := 0;
   Buffer[6].Codigo := '';
   Buffer[6].Fecha_1.Ano := 0;
   Buffer[6].Fecha_1.Mes := 0;
   Buffer[6].Fecha_1.Dia := 0;
   Buffer[6].Fecha_1.DiaSemana := 0;
   Buffer[6].Fecha_1.Hora := 0;
   Buffer[6].Fecha_1.Minuto := 0;
   Buffer[6].Fecha_1.Segundo := 0;
   Buffer[6].Fecha_1.NanoSegundo := 0;
   Buffer[6].Fecha_2.Ano := 0;
   Buffer[6].Fecha_2.Mes := 0;
   Buffer[6].Fecha_2.Dia := 0;
   Buffer[6].Fecha_2.DiaSemana := 0;
   Buffer[6].Fecha_2.Hora := 0;
   Buffer[6].Fecha_2.Minuto := 0;
   Buffer[6].Fecha_2.Segundo := 0;
   Buffer[6].Fecha_2.NanoSegundo := 0;
   Buffer[6].Fecha_3.Ano := 0;
   Buffer[6].Fecha_3.Mes := 0;
   Buffer[6].Fecha_3.Dia := 0;
   Buffer[6].Fecha_3.DiaSemana := 0;
   Buffer[6].Fecha_3.Hora := 0;
   Buffer[6].Fecha_3.Minuto := 0;
   Buffer[6].Fecha_3.Segundo := 0;
   Buffer[6].Fecha_3.NanoSegundo := 0;
   Buffer[6].String_1 := '';
   Buffer[6].String_2 := '';
   Buffer[6].String_3 := '';
   Buffer[6].String_4 := '';
   Buffer[6].String_5 := '';
   Buffer[6].String_6 := '';
   Buffer[6].String_7 := '';
   Buffer[6].String_8 := '';
   Buffer[6].String_9 := '';
   Buffer[6].String_10 := '';
   Buffer[6].Bool_1 := FALSE;
   Buffer[6].Bool_2 := FALSE;
   Buffer[6].Bool_3 := FALSE;
   Buffer[6].Bool_4 := FALSE;
   Buffer[6].Bool_5 := FALSE;
   Buffer[6].Bool_6 := FALSE;
   Buffer[6].Bool_7 := FALSE;
   Buffer[6].Bool_8 := FALSE;
   Buffer[6].Bool_9 := FALSE;
   Buffer[6].Bool_10 := FALSE;
   Buffer[6].Bool_11 := FALSE;
   Buffer[6].Bool_12 := FALSE;
   Buffer[6].Bool_13 := FALSE;
   Buffer[6].Bool_14 := FALSE;
   Buffer[6].Bool_15 := FALSE;
   Buffer[6].Bool_16 := FALSE;
   Buffer[6].Bool_17 := FALSE;
   Buffer[6].Bool_18 := FALSE;
   Buffer[6].Bool_19 := FALSE;
   Buffer[6].Bool_20 := FALSE;
   Buffer[6].Bool_21 := FALSE;
   Buffer[6].Bool_22 := FALSE;
   Buffer[6].Bool_23 := FALSE;
   Buffer[6].Bool_24 := FALSE;
   Buffer[6].Bool_25 := FALSE;
   Buffer[6].Bool_26 := FALSE;
   Buffer[6].Bool_27 := FALSE;
   Buffer[6].Bool_28 := FALSE;
   Buffer[6].Bool_29 := FALSE;
   Buffer[6].Bool_30 := FALSE;
   Buffer[6].Bool_31 := FALSE;
   Buffer[6].Bool_32 := FALSE;
   Buffer[6].Real_1 := 0.0;
   Buffer[6].Real_2 := 0.0;
   Buffer[6].Real_3 := 0.0;
   Buffer[6].Real_4 := 0.0;
   Buffer[6].Real_5 := 0.0;
   Buffer[6].Real_6 := 0.0;
   Buffer[6].Real_7 := 0.0;
   Buffer[6].Real_8 := 0.0;
   Buffer[6].Real_9 := 0.0;
   Buffer[6].Real_10 := 0.0;
   Buffer[6].Real_11 := 0.0;
   Buffer[6].Real_12 := 0.0;
   Buffer[6].Real_13 := 0.0;
   Buffer[6].Real_14 := 0.0;
   Buffer[6].Real_15 := 0.0;
   Buffer[6].Real_16 := 0.0;
   Buffer[6].Real_17 := 0.0;
   Buffer[6].Real_18 := 0.0;
   Buffer[6].Real_19 := 0.0;
   Buffer[6].Real_20 := 0.0;
   Buffer[6].Int_1 := 0;
   Buffer[6].Int_2 := 0;
   Buffer[6].Int_3 := 0;
   Buffer[6].Int_4 := 0;
   Buffer[6].Int_5 := 0;
   Buffer[6].Int_6 := 0;
   Buffer[6].Int_7 := 0;
   Buffer[6].Int_8 := 0;
   Buffer[6].Int_9 := 0;
   Buffer[6].Int_10 := 0;
   Buffer[6].Int_11 := 0;
   Buffer[6].Int_12 := 0;
   Buffer[6].Int_13 := 0;
   Buffer[6].Int_14 := 0;
   Buffer[6].Int_15 := 0;
   Buffer[6].Int_16 := 0;
   Buffer[6].Int_17 := 0;
   Buffer[6].Int_18 := 0;
   Buffer[6].Int_19 := 0;
   Buffer[6].Int_20 := 0;
   Buffer[7].Registrar := 0;
   Buffer[7].Id := '';
   Buffer[7].Tipo := 0;
   Buffer[7].Codigo := '';
   Buffer[7].Fecha_1.Ano := 0;
   Buffer[7].Fecha_1.Mes := 0;
   Buffer[7].Fecha_1.Dia := 0;
   Buffer[7].Fecha_1.DiaSemana := 0;
   Buffer[7].Fecha_1.Hora := 0;
   Buffer[7].Fecha_1.Minuto := 0;
   Buffer[7].Fecha_1.Segundo := 0;
   Buffer[7].Fecha_1.NanoSegundo := 0;
   Buffer[7].Fecha_2.Ano := 0;
   Buffer[7].Fecha_2.Mes := 0;
   Buffer[7].Fecha_2.Dia := 0;
   Buffer[7].Fecha_2.DiaSemana := 0;
   Buffer[7].Fecha_2.Hora := 0;
   Buffer[7].Fecha_2.Minuto := 0;
   Buffer[7].Fecha_2.Segundo := 0;
   Buffer[7].Fecha_2.NanoSegundo := 0;
   Buffer[7].Fecha_3.Ano := 0;
   Buffer[7].Fecha_3.Mes := 0;
   Buffer[7].Fecha_3.Dia := 0;
   Buffer[7].Fecha_3.DiaSemana := 0;
   Buffer[7].Fecha_3.Hora := 0;
   Buffer[7].Fecha_3.Minuto := 0;
   Buffer[7].Fecha_3.Segundo := 0;
   Buffer[7].Fecha_3.NanoSegundo := 0;
   Buffer[7].String_1 := '';
   Buffer[7].String_2 := '';
   Buffer[7].String_3 := '';
   Buffer[7].String_4 := '';
   Buffer[7].String_5 := '';
   Buffer[7].String_6 := '';
   Buffer[7].String_7 := '';
   Buffer[7].String_8 := '';
   Buffer[7].String_9 := '';
   Buffer[7].String_10 := '';
   Buffer[7].Bool_1 := FALSE;
   Buffer[7].Bool_2 := FALSE;
   Buffer[7].Bool_3 := FALSE;
   Buffer[7].Bool_4 := FALSE;
   Buffer[7].Bool_5 := FALSE;
   Buffer[7].Bool_6 := FALSE;
   Buffer[7].Bool_7 := FALSE;
   Buffer[7].Bool_8 := FALSE;
   Buffer[7].Bool_9 := FALSE;
   Buffer[7].Bool_10 := FALSE;
   Buffer[7].Bool_11 := FALSE;
   Buffer[7].Bool_12 := FALSE;
   Buffer[7].Bool_13 := FALSE;
   Buffer[7].Bool_14 := FALSE;
   Buffer[7].Bool_15 := FALSE;
   Buffer[7].Bool_16 := FALSE;
   Buffer[7].Bool_17 := FALSE;
   Buffer[7].Bool_18 := FALSE;
   Buffer[7].Bool_19 := FALSE;
   Buffer[7].Bool_20 := FALSE;
   Buffer[7].Bool_21 := FALSE;
   Buffer[7].Bool_22 := FALSE;
   Buffer[7].Bool_23 := FALSE;
   Buffer[7].Bool_24 := FALSE;
   Buffer[7].Bool_25 := FALSE;
   Buffer[7].Bool_26 := FALSE;
   Buffer[7].Bool_27 := FALSE;
   Buffer[7].Bool_28 := FALSE;
   Buffer[7].Bool_29 := FALSE;
   Buffer[7].Bool_30 := FALSE;
   Buffer[7].Bool_31 := FALSE;
   Buffer[7].Bool_32 := FALSE;
   Buffer[7].Real_1 := 0.0;
   Buffer[7].Real_2 := 0.0;
   Buffer[7].Real_3 := 0.0;
   Buffer[7].Real_4 := 0.0;
   Buffer[7].Real_5 := 0.0;
   Buffer[7].Real_6 := 0.0;
   Buffer[7].Real_7 := 0.0;
   Buffer[7].Real_8 := 0.0;
   Buffer[7].Real_9 := 0.0;
   Buffer[7].Real_10 := 0.0;
   Buffer[7].Real_11 := 0.0;
   Buffer[7].Real_12 := 0.0;
   Buffer[7].Real_13 := 0.0;
   Buffer[7].Real_14 := 0.0;
   Buffer[7].Real_15 := 0.0;
   Buffer[7].Real_16 := 0.0;
   Buffer[7].Real_17 := 0.0;
   Buffer[7].Real_18 := 0.0;
   Buffer[7].Real_19 := 0.0;
   Buffer[7].Real_20 := 0.0;
   Buffer[7].Int_1 := 0;
   Buffer[7].Int_2 := 0;
   Buffer[7].Int_3 := 0;
   Buffer[7].Int_4 := 0;
   Buffer[7].Int_5 := 0;
   Buffer[7].Int_6 := 0;
   Buffer[7].Int_7 := 0;
   Buffer[7].Int_8 := 0;
   Buffer[7].Int_9 := 0;
   Buffer[7].Int_10 := 0;
   Buffer[7].Int_11 := 0;
   Buffer[7].Int_12 := 0;
   Buffer[7].Int_13 := 0;
   Buffer[7].Int_14 := 0;
   Buffer[7].Int_15 := 0;
   Buffer[7].Int_16 := 0;
   Buffer[7].Int_17 := 0;
   Buffer[7].Int_18 := 0;
   Buffer[7].Int_19 := 0;
   Buffer[7].Int_20 := 0;
   Buffer[8].Registrar := 0;
   Buffer[8].Id := '';
   Buffer[8].Tipo := 0;
   Buffer[8].Codigo := '';
   Buffer[8].Fecha_1.Ano := 0;
   Buffer[8].Fecha_1.Mes := 0;
   Buffer[8].Fecha_1.Dia := 0;
   Buffer[8].Fecha_1.DiaSemana := 0;
   Buffer[8].Fecha_1.Hora := 0;
   Buffer[8].Fecha_1.Minuto := 0;
   Buffer[8].Fecha_1.Segundo := 0;
   Buffer[8].Fecha_1.NanoSegundo := 0;
   Buffer[8].Fecha_2.Ano := 0;
   Buffer[8].Fecha_2.Mes := 0;
   Buffer[8].Fecha_2.Dia := 0;
   Buffer[8].Fecha_2.DiaSemana := 0;
   Buffer[8].Fecha_2.Hora := 0;
   Buffer[8].Fecha_2.Minuto := 0;
   Buffer[8].Fecha_2.Segundo := 0;
   Buffer[8].Fecha_2.NanoSegundo := 0;
   Buffer[8].Fecha_3.Ano := 0;
   Buffer[8].Fecha_3.Mes := 0;
   Buffer[8].Fecha_3.Dia := 0;
   Buffer[8].Fecha_3.DiaSemana := 0;
   Buffer[8].Fecha_3.Hora := 0;
   Buffer[8].Fecha_3.Minuto := 0;
   Buffer[8].Fecha_3.Segundo := 0;
   Buffer[8].Fecha_3.NanoSegundo := 0;
   Buffer[8].String_1 := '';
   Buffer[8].String_2 := '';
   Buffer[8].String_3 := '';
   Buffer[8].String_4 := '';
   Buffer[8].String_5 := '';
   Buffer[8].String_6 := '';
   Buffer[8].String_7 := '';
   Buffer[8].String_8 := '';
   Buffer[8].String_9 := '';
   Buffer[8].String_10 := '';
   Buffer[8].Bool_1 := FALSE;
   Buffer[8].Bool_2 := FALSE;
   Buffer[8].Bool_3 := FALSE;
   Buffer[8].Bool_4 := FALSE;
   Buffer[8].Bool_5 := FALSE;
   Buffer[8].Bool_6 := FALSE;
   Buffer[8].Bool_7 := FALSE;
   Buffer[8].Bool_8 := FALSE;
   Buffer[8].Bool_9 := FALSE;
   Buffer[8].Bool_10 := FALSE;
   Buffer[8].Bool_11 := FALSE;
   Buffer[8].Bool_12 := FALSE;
   Buffer[8].Bool_13 := FALSE;
   Buffer[8].Bool_14 := FALSE;
   Buffer[8].Bool_15 := FALSE;
   Buffer[8].Bool_16 := FALSE;
   Buffer[8].Bool_17 := FALSE;
   Buffer[8].Bool_18 := FALSE;
   Buffer[8].Bool_19 := FALSE;
   Buffer[8].Bool_20 := FALSE;
   Buffer[8].Bool_21 := FALSE;
   Buffer[8].Bool_22 := FALSE;
   Buffer[8].Bool_23 := FALSE;
   Buffer[8].Bool_24 := FALSE;
   Buffer[8].Bool_25 := FALSE;
   Buffer[8].Bool_26 := FALSE;
   Buffer[8].Bool_27 := FALSE;
   Buffer[8].Bool_28 := FALSE;
   Buffer[8].Bool_29 := FALSE;
   Buffer[8].Bool_30 := FALSE;
   Buffer[8].Bool_31 := FALSE;
   Buffer[8].Bool_32 := FALSE;
   Buffer[8].Real_1 := 0.0;
   Buffer[8].Real_2 := 0.0;
   Buffer[8].Real_3 := 0.0;
   Buffer[8].Real_4 := 0.0;
   Buffer[8].Real_5 := 0.0;
   Buffer[8].Real_6 := 0.0;
   Buffer[8].Real_7 := 0.0;
   Buffer[8].Real_8 := 0.0;
   Buffer[8].Real_9 := 0.0;
   Buffer[8].Real_10 := 0.0;
   Buffer[8].Real_11 := 0.0;
   Buffer[8].Real_12 := 0.0;
   Buffer[8].Real_13 := 0.0;
   Buffer[8].Real_14 := 0.0;
   Buffer[8].Real_15 := 0.0;
   Buffer[8].Real_16 := 0.0;
   Buffer[8].Real_17 := 0.0;
   Buffer[8].Real_18 := 0.0;
   Buffer[8].Real_19 := 0.0;
   Buffer[8].Real_20 := 0.0;
   Buffer[8].Int_1 := 0;
   Buffer[8].Int_2 := 0;
   Buffer[8].Int_3 := 0;
   Buffer[8].Int_4 := 0;
   Buffer[8].Int_5 := 0;
   Buffer[8].Int_6 := 0;
   Buffer[8].Int_7 := 0;
   Buffer[8].Int_8 := 0;
   Buffer[8].Int_9 := 0;
   Buffer[8].Int_10 := 0;
   Buffer[8].Int_11 := 0;
   Buffer[8].Int_12 := 0;
   Buffer[8].Int_13 := 0;
   Buffer[8].Int_14 := 0;
   Buffer[8].Int_15 := 0;
   Buffer[8].Int_16 := 0;
   Buffer[8].Int_17 := 0;
   Buffer[8].Int_18 := 0;
   Buffer[8].Int_19 := 0;
   Buffer[8].Int_20 := 0;
   Buffer[9].Registrar := 0;
   Buffer[9].Id := '';
   Buffer[9].Tipo := 0;
   Buffer[9].Codigo := '';
   Buffer[9].Fecha_1.Ano := 0;
   Buffer[9].Fecha_1.Mes := 0;
   Buffer[9].Fecha_1.Dia := 0;
   Buffer[9].Fecha_1.DiaSemana := 0;
   Buffer[9].Fecha_1.Hora := 0;
   Buffer[9].Fecha_1.Minuto := 0;
   Buffer[9].Fecha_1.Segundo := 0;
   Buffer[9].Fecha_1.NanoSegundo := 0;
   Buffer[9].Fecha_2.Ano := 0;
   Buffer[9].Fecha_2.Mes := 0;
   Buffer[9].Fecha_2.Dia := 0;
   Buffer[9].Fecha_2.DiaSemana := 0;
   Buffer[9].Fecha_2.Hora := 0;
   Buffer[9].Fecha_2.Minuto := 0;
   Buffer[9].Fecha_2.Segundo := 0;
   Buffer[9].Fecha_2.NanoSegundo := 0;
   Buffer[9].Fecha_3.Ano := 0;
   Buffer[9].Fecha_3.Mes := 0;
   Buffer[9].Fecha_3.Dia := 0;
   Buffer[9].Fecha_3.DiaSemana := 0;
   Buffer[9].Fecha_3.Hora := 0;
   Buffer[9].Fecha_3.Minuto := 0;
   Buffer[9].Fecha_3.Segundo := 0;
   Buffer[9].Fecha_3.NanoSegundo := 0;
   Buffer[9].String_1 := '';
   Buffer[9].String_2 := '';
   Buffer[9].String_3 := '';
   Buffer[9].String_4 := '';
   Buffer[9].String_5 := '';
   Buffer[9].String_6 := '';
   Buffer[9].String_7 := '';
   Buffer[9].String_8 := '';
   Buffer[9].String_9 := '';
   Buffer[9].String_10 := '';
   Buffer[9].Bool_1 := FALSE;
   Buffer[9].Bool_2 := FALSE;
   Buffer[9].Bool_3 := FALSE;
   Buffer[9].Bool_4 := FALSE;
   Buffer[9].Bool_5 := FALSE;
   Buffer[9].Bool_6 := FALSE;
   Buffer[9].Bool_7 := FALSE;
   Buffer[9].Bool_8 := FALSE;
   Buffer[9].Bool_9 := FALSE;
   Buffer[9].Bool_10 := FALSE;
   Buffer[9].Bool_11 := FALSE;
   Buffer[9].Bool_12 := FALSE;
   Buffer[9].Bool_13 := FALSE;
   Buffer[9].Bool_14 := FALSE;
   Buffer[9].Bool_15 := FALSE;
   Buffer[9].Bool_16 := FALSE;
   Buffer[9].Bool_17 := FALSE;
   Buffer[9].Bool_18 := FALSE;
   Buffer[9].Bool_19 := FALSE;
   Buffer[9].Bool_20 := FALSE;
   Buffer[9].Bool_21 := FALSE;
   Buffer[9].Bool_22 := FALSE;
   Buffer[9].Bool_23 := FALSE;
   Buffer[9].Bool_24 := FALSE;
   Buffer[9].Bool_25 := FALSE;
   Buffer[9].Bool_26 := FALSE;
   Buffer[9].Bool_27 := FALSE;
   Buffer[9].Bool_28 := FALSE;
   Buffer[9].Bool_29 := FALSE;
   Buffer[9].Bool_30 := FALSE;
   Buffer[9].Bool_31 := FALSE;
   Buffer[9].Bool_32 := FALSE;
   Buffer[9].Real_1 := 0.0;
   Buffer[9].Real_2 := 0.0;
   Buffer[9].Real_3 := 0.0;
   Buffer[9].Real_4 := 0.0;
   Buffer[9].Real_5 := 0.0;
   Buffer[9].Real_6 := 0.0;
   Buffer[9].Real_7 := 0.0;
   Buffer[9].Real_8 := 0.0;
   Buffer[9].Real_9 := 0.0;
   Buffer[9].Real_10 := 0.0;
   Buffer[9].Real_11 := 0.0;
   Buffer[9].Real_12 := 0.0;
   Buffer[9].Real_13 := 0.0;
   Buffer[9].Real_14 := 0.0;
   Buffer[9].Real_15 := 0.0;
   Buffer[9].Real_16 := 0.0;
   Buffer[9].Real_17 := 0.0;
   Buffer[9].Real_18 := 0.0;
   Buffer[9].Real_19 := 0.0;
   Buffer[9].Real_20 := 0.0;
   Buffer[9].Int_1 := 0;
   Buffer[9].Int_2 := 0;
   Buffer[9].Int_3 := 0;
   Buffer[9].Int_4 := 0;
   Buffer[9].Int_5 := 0;
   Buffer[9].Int_6 := 0;
   Buffer[9].Int_7 := 0;
   Buffer[9].Int_8 := 0;
   Buffer[9].Int_9 := 0;
   Buffer[9].Int_10 := 0;
   Buffer[9].Int_11 := 0;
   Buffer[9].Int_12 := 0;
   Buffer[9].Int_13 := 0;
   Buffer[9].Int_14 := 0;
   Buffer[9].Int_15 := 0;
   Buffer[9].Int_16 := 0;
   Buffer[9].Int_17 := 0;
   Buffer[9].Int_18 := 0;
   Buffer[9].Int_19 := 0;
   Buffer[9].Int_20 := 0;
   Buffer[10].Registrar := 0;
   Buffer[10].Id := '';
   Buffer[10].Tipo := 0;
   Buffer[10].Codigo := '';
   Buffer[10].Fecha_1.Ano := 0;
   Buffer[10].Fecha_1.Mes := 0;
   Buffer[10].Fecha_1.Dia := 0;
   Buffer[10].Fecha_1.DiaSemana := 0;
   Buffer[10].Fecha_1.Hora := 0;
   Buffer[10].Fecha_1.Minuto := 0;
   Buffer[10].Fecha_1.Segundo := 0;
   Buffer[10].Fecha_1.NanoSegundo := 0;
   Buffer[10].Fecha_2.Ano := 0;
   Buffer[10].Fecha_2.Mes := 0;
   Buffer[10].Fecha_2.Dia := 0;
   Buffer[10].Fecha_2.DiaSemana := 0;
   Buffer[10].Fecha_2.Hora := 0;
   Buffer[10].Fecha_2.Minuto := 0;
   Buffer[10].Fecha_2.Segundo := 0;
   Buffer[10].Fecha_2.NanoSegundo := 0;
   Buffer[10].Fecha_3.Ano := 0;
   Buffer[10].Fecha_3.Mes := 0;
   Buffer[10].Fecha_3.Dia := 0;
   Buffer[10].Fecha_3.DiaSemana := 0;
   Buffer[10].Fecha_3.Hora := 0;
   Buffer[10].Fecha_3.Minuto := 0;
   Buffer[10].Fecha_3.Segundo := 0;
   Buffer[10].Fecha_3.NanoSegundo := 0;
   Buffer[10].String_1 := '';
   Buffer[10].String_2 := '';
   Buffer[10].String_3 := '';
   Buffer[10].String_4 := '';
   Buffer[10].String_5 := '';
   Buffer[10].String_6 := '';
   Buffer[10].String_7 := '';
   Buffer[10].String_8 := '';
   Buffer[10].String_9 := '';
   Buffer[10].String_10 := '';
   Buffer[10].Bool_1 := FALSE;
   Buffer[10].Bool_2 := FALSE;
   Buffer[10].Bool_3 := FALSE;
   Buffer[10].Bool_4 := FALSE;
   Buffer[10].Bool_5 := FALSE;
   Buffer[10].Bool_6 := FALSE;
   Buffer[10].Bool_7 := FALSE;
   Buffer[10].Bool_8 := FALSE;
   Buffer[10].Bool_9 := FALSE;
   Buffer[10].Bool_10 := FALSE;
   Buffer[10].Bool_11 := FALSE;
   Buffer[10].Bool_12 := FALSE;
   Buffer[10].Bool_13 := FALSE;
   Buffer[10].Bool_14 := FALSE;
   Buffer[10].Bool_15 := FALSE;
   Buffer[10].Bool_16 := FALSE;
   Buffer[10].Bool_17 := FALSE;
   Buffer[10].Bool_18 := FALSE;
   Buffer[10].Bool_19 := FALSE;
   Buffer[10].Bool_20 := FALSE;
   Buffer[10].Bool_21 := FALSE;
   Buffer[10].Bool_22 := FALSE;
   Buffer[10].Bool_23 := FALSE;
   Buffer[10].Bool_24 := FALSE;
   Buffer[10].Bool_25 := FALSE;
   Buffer[10].Bool_26 := FALSE;
   Buffer[10].Bool_27 := FALSE;
   Buffer[10].Bool_28 := FALSE;
   Buffer[10].Bool_29 := FALSE;
   Buffer[10].Bool_30 := FALSE;
   Buffer[10].Bool_31 := FALSE;
   Buffer[10].Bool_32 := FALSE;
   Buffer[10].Real_1 := 0.0;
   Buffer[10].Real_2 := 0.0;
   Buffer[10].Real_3 := 0.0;
   Buffer[10].Real_4 := 0.0;
   Buffer[10].Real_5 := 0.0;
   Buffer[10].Real_6 := 0.0;
   Buffer[10].Real_7 := 0.0;
   Buffer[10].Real_8 := 0.0;
   Buffer[10].Real_9 := 0.0;
   Buffer[10].Real_10 := 0.0;
   Buffer[10].Real_11 := 0.0;
   Buffer[10].Real_12 := 0.0;
   Buffer[10].Real_13 := 0.0;
   Buffer[10].Real_14 := 0.0;
   Buffer[10].Real_15 := 0.0;
   Buffer[10].Real_16 := 0.0;
   Buffer[10].Real_17 := 0.0;
   Buffer[10].Real_18 := 0.0;
   Buffer[10].Real_19 := 0.0;
   Buffer[10].Real_20 := 0.0;
   Buffer[10].Int_1 := 0;
   Buffer[10].Int_2 := 0;
   Buffer[10].Int_3 := 0;
   Buffer[10].Int_4 := 0;
   Buffer[10].Int_5 := 0;
   Buffer[10].Int_6 := 0;
   Buffer[10].Int_7 := 0;
   Buffer[10].Int_8 := 0;
   Buffer[10].Int_9 := 0;
   Buffer[10].Int_10 := 0;
   Buffer[10].Int_11 := 0;
   Buffer[10].Int_12 := 0;
   Buffer[10].Int_13 := 0;
   Buffer[10].Int_14 := 0;
   Buffer[10].Int_15 := 0;
   Buffer[10].Int_16 := 0;
   Buffer[10].Int_17 := 0;
   Buffer[10].Int_18 := 0;
   Buffer[10].Int_19 := 0;
   Buffer[10].Int_20 := 0;

END_DATA_BLOCK

